ABB RobotStudio station: COLISIONYOGUR.rspag

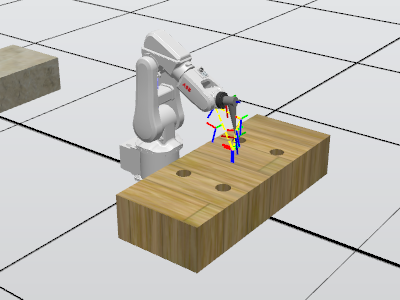
--- station ---
Station Project1 (saved by RobotStudio 25.3.11371.0)
Controller IRB120_3_58
  mechanical unit ROB_1: IRB120_3_58__01, 6 joints, base frame (0, 0, 0) mm
Layout (positions relative to the parent item):
  - IRB120_3_58__01 [mechanism, from %ABB.RobotStudio.Models.IRB120%\IRB120_3_58_G_01.rslib] at (0, 0, 0) mm; joint values [0, -0.0079, 0.5429, 0, -0.6884, 0] (rad or m)
  - ventosa [mechanism] at (364.51, 0, 477.22) mm, rotated rx 0 ry 81.21 rz 0 deg
      TCP ventosa at (160, 0, 30) mm, rotated rx 0 ry 90 rz 0 deg
      links: ventosa
  - mesa [part] at (-1400, 0, 0) mm, size 400 x 1000 x 200 mm
  - yogur [smart component]
      signals: DI sacarYogur, DO colision, DI ventosa
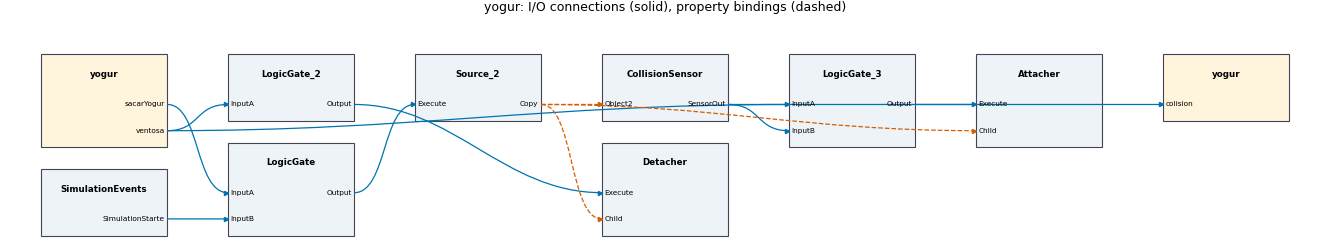
      connections:
        CollisionSensor.SensorOut -> yogur.colision
        yogur.sacarYogur -> LogicGate.InputA
        SimulationEvents.SimulationStarted -> LogicGate.InputB
        LogicGate.Output -> Source_2.Execute
        yogur.ventosa -> LogicGate_2.InputA
        LogicGate_2.Output -> Detacher.Execute
        yogur.ventosa -> LogicGate_3.InputA
        CollisionSensor.SensorOut -> LogicGate_3.InputB
        LogicGate_3.Output -> Attacher.Execute
        Source_2.Copy => CollisionSensor.Object2
        Source_2.Copy => Detacher.Child
        Source_2.Copy => Attacher.Child
    - yogur [part], size 60 x 80 x 72 mm
    - Source_2 [smart component, from Components\Source.rslib]
        properties: Source=yogur; Copy=(none); Parent=(none); Position=[0.4 0 0.21]; Orientation=[0 0 0]; Transient=true; PhysicsBehavior=3
    - CollisionSensor [smart component, from Components\CollisionSensor.rslib]
        properties: Object1=ventosa; Object2=(none); NearMiss=0; Part1=(none); Part2=(none); CollisionType=0
    - LogicGate [smart component, from Components\LogicGate.rslib]
        properties: Operator=OR; Delay=0
    - SimulationEvents [smart component, from Components\SimulationEvents.rslib]
    - LogicGate_2 [smart component, from Components\LogicGate.rslib]
        properties: Operator=NOT; Delay=0
    - Attacher [smart component, from Components\Attacher.rslib]
        properties: Parent=ventosa; Flange=0; Child=(none); Mount=false; Offset=[0 0 0]; Orientation=[0 0 0]
    - Detacher [smart component, from Components\Detacher.rslib]
        properties: Child=(none); KeepPosition=true
    - LogicGate_3 [smart component, from Components\LogicGate.rslib]
        properties: Operator=AND; Delay=0
  - Pieza_15 [part] at (0.02, -0.01, 3.79) mm, size 400 x 1000 x 200 mm
Attachment: ventosa is attached to IRB120_3_58__01 / Link6
Attachment: Source_2 is attached to Detacher
Station logic (signal -> signal, property => property):
  IRB120_3_58.DO_0 -> yogur.ventosa
  yogur.colision -> IRB120_3_58.DI_0

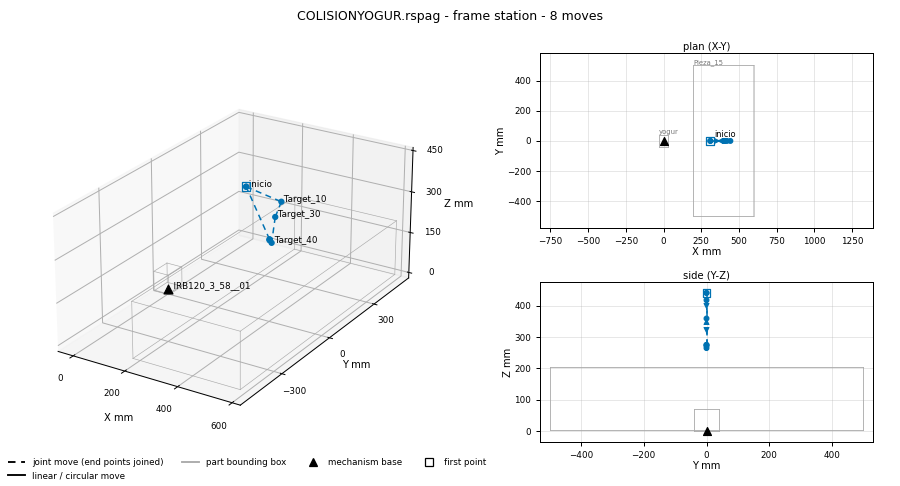
[picture p0: tool path of COLISIONYOGUR.rspag in frame station, 8 of 8 moves have a stored position in this frame; points joined in program order, loops and branches not executed]
--- Controller Data/IRB120_3_58/RAPID/TASK1/PROGMOD/CalibData.mod ---
MODULE CalibData
    PERS tooldata ventosa:=[TRUE,[[160,0,30],[0.707107,0,0.707107,0]],[1,[0,0,1],[1,0,0,0],0,0,0]];
    TASK PERS wobjdata Workobject_1:=[FALSE,TRUE,"",[[0,0,0],[1,0,0,0]],[[0,0,0],[1,0,0,0]]];
ENDMODULE

--- Controller Data/IRB120_3_58/RAPID/TASK1/PROGMOD/Module1.mod ---
MODULE Module1
    CONST robtarget inicio:=[[310.334591186,0,440.435935394],[0.258819045,0,-0.965925826,0],[0,0,0,0],[9E+09,9E+09,9E+09,9E+09,9E+09,9E+09]];
    CONST robtarget yogur:=[[400.000016072,0,272],[0,0,1,0],[0,0,0,1],[9E+09,9E+09,9E+09,9E+09,9E+09,9E+09]];
    CONST robtarget yogur_1:=[[400,0,275],[0,0,1,0],[0,0,0,1],[9E+09,9E+09,9E+09,9E+09,9E+09,9E+09]];
    CONST robtarget Target_10:=[[443.415150227,0,417.419464125],[0.022577684,0,-0.999745092,0],[0,0,0,1],[9E+09,9E+09,9E+09,9E+09,9E+09,9E+09]];
    CONST robtarget Target_20:=[[315.695646104,0,340.576081201],[0.11811315,0,-0.993000143,0],[0,0,0,1],[9E+09,9E+09,9E+09,9E+09,9E+09,9E+09]];
    CONST robtarget Target_30:=[[420.848371875,0,358.973880322],[0.118113043,0,0.993000156,0],[0,0,0,1],[9E+09,9E+09,9E+09,9E+09,9E+09,9E+09]];
    CONST robtarget Target_40:=[[407.925787387,0,264.736188054],[0.00488199,0,0.999988083,0],[0,0,0,1],[9E+09,9E+09,9E+09,9E+09,9E+09,9E+09]];
    !***********************************************************
    !
    ! M?dulo:  Module1
    !
    ! Descripción:
    !   <Introduzca la descripción aquí>
    !
    ! Autor: ferna
    !
    ! Versión: 1.0
    !
    !***********************************************************


    !***********************************************************
    !
    ! Procedimiento Main
    !
    !   Este es el punto de entrada de su programa
    !
    !***********************************************************
    PROC main()
        !Add your code here
        Path_10;
    ENDPROC
    PROC Path_10()
        MoveJ inicio,v150,z100,ventosa\WObj:=Workobject_1;
        MoveJ Target_10,v1000,z100,ventosa\WObj:=Workobject_1;
        MoveJ Target_30,v1000,z100,ventosa\WObj:=Workobject_1;
        MoveJ Target_40,v100,z100,ventosa\WObj:=Workobject_1;
        MoveJ yogur_1,v100,z10,ventosa\WObj:=Workobject_1;
        WaitTime 1;
        MoveLDO yogur,v100,z0,ventosa\WObj:=Workobject_1, DO_0,1;
        MoveL yogur_1,v100,z0,ventosa\WObj:=Workobject_1;


        MoveJ inicio,v150,z100,ventosa\WObj:=Workobject_1;
              WaitTime 1;
        RESET DO_0;
    ENDPROC
ENDMODULE

--- Controller Data/IRB120_3_58/SYSPAR/EIO.cfg ---
EIO:CFG_1.0:6:1::
#
INDUSTRIAL_NETWORK:

      -Name "DeviceNet" -Label "DeviceNet Master/Slave Network" -Address "2"
#
DEVICENET_DEVICE:

      -Name "d652" -VendorName "ABB Robotics" -ProductName "24 VDC I/O Device"\
      -Label "DSQC 652 24 VDC I/O Device" -Address 10 -ProductCode 26\
      -DeviceType 7 -ConnectionType "COS" -OutputSize 2 -InputSize 2
#
DEVICENET_INTERNAL_DEVICE:

      -Name "DN_Internal_Device" -VendorName "ABB Robotics"\
      -ProductName "DeviceNet Internal Slave Device"
#
EIO_SIGNAL:

      -Name "DI_0" -SignalType "DI" -Device "d652" -DeviceMap "0" -Access "All"

      -Name "DI_1" -SignalType "DI" -Device "d652" -DeviceMap "1" -Access "All"

      -Name "DI_2" -SignalType "DI" -Device "d652" -DeviceMap "2" -Access "All"

      -Name "DI_3" -SignalType "DI" -Device "d652" -DeviceMap "3" -Access "All"

      -Name "DO_3" -SignalType "DO" -Device "d652" -DeviceMap "3" -Access "All"

      -Name "DO_2" -SignalType "DO" -Device "d652" -DeviceMap "2" -Access "All"

      -Name "DO_0" -SignalType "DO" -Device "d652" -DeviceMap "0" -Access "All"
